FUNCTION_BLOCK HaltBehaviour IMPLEMENTS I_Task, I_Cyclic, I_Abortable, I_Object
VAR_INPUT
END_VAR
VAR_OUTPUT
END_VAR
VAR
	mcHalt : Tc2_MC2.MC_Halt;
	_Axis : REFERENCE TO Tc2_MC2.AXIS_REF;
END_VAR

{analysis -2}

METHOD Abort : HRESULT
mcHalt.Execute := FALSE;
END_METHOD

PROPERTY AxisRef : reference to Axis_Ref
GET // PUBLIC
AxisRef REF= _Axis;
END_GET
SET
_Axis REF= AxisRef;
END_SET
END_PROPERTY

PROPERTY Busy : BOOL
GET
Busy := mcHalt.Busy;
END_GET
END_PROPERTY

METHOD Cycle : HRESULT
VAR_INPUT
END_VAR
mcHalt(Axis := _Axis);
mcHalt.Execute := FALSE;
END_METHOD

PROPERTY Deceleration : MC_LREAL
GET
Deceleration := mcHalt.Deceleration;
END_GET
SET
IF Deceleration >= 0.0 THEN
	mcHalt.Deceleration := Deceleration;
END_IF
END_SET
END_PROPERTY

PROPERTY Done : BOOL
GET
Done := mcHalt.Done;
END_GET
END_PROPERTY

PROPERTY Error : BOOL
GET
Error := mcHalt.Error;
END_GET
END_PROPERTY

METHOD Execute : HRESULT
VAR_INPUT
END_VAR
IF _Axis.Status.Moving AND NOT mcHalt.Busy THEN
	Execute := S_OK;
	mcHalt.Execute := TRUE;
ELSE
	Execute := S_FALSE;
END_IF
END_METHOD

PROPERTY Jerk : MC_LREAL
GET
Jerk := mcHalt.Jerk;
END_GET
SET
IF Jerk >= 0.0 THEN
	mcHalt.Jerk := Jerk;
END_IF
END_SET
END_PROPERTY

METHOD RegisterWithParent
VAR_INPUT
	Runner	: I_HostObjects;
END_VAR
Runner.RegisterAbortable(THIS^);
Runner.RegisterCyclic(THIS^);
Runner.RegisterTask(THIS^);
END_METHOD

END_FUNCTION_BLOCK

(* stored: Version 1.1.0.1
   POU HaltBehaviour: Id {8f902aee-94bf-4385-bdcf-ca790f894752}, SpecialFunc None
   Method Abort: Id {628339b1-4bd1-432e-8277-d60f3e75db0d}
   Property AxisRef: Id {1eac54a6-2798-4751-837f-d3da316af4f3}
   Get Get: Id {b1c4cfd8-893a-485e-bd47-04ef2d23093f}
   Set Set: Id {4a81d8e2-63e1-4eb7-82a1-2f62a4d2f98c}
   Property Busy: Id {372dcfaa-8cbd-4cb0-a70e-bb4041d8e255}
   Get Get: Id {91d2b55e-e06d-4906-afcd-b4c07ffa30db}
   Method Cycle: Id {82fe1e7b-ab2b-4a89-9b59-5eb25d835959}
   Property Deceleration: Id {268ed3d1-2986-429d-85cd-2c570b60d9d7}
   Get Get: Id {907709a1-b0ba-4945-8711-6554db8f1dc0}
   Set Set: Id {502b45a2-e349-483e-b36a-b0db162a9224}
   Property Done: Id {0d4d59d1-0a33-4a35-91db-70cde82f5006}
   Get Get: Id {5c83bea7-d010-40d8-bc69-060934607785}
   Property Error: Id {3e7959eb-71d7-4ee5-89e9-4dd47b034681}
   Get Get: Id {1eaeb28a-b2d3-41f6-9d16-23d88d0071e2}
   Method Execute: Id {020a5dad-2d55-4c66-8489-dc08945209ce}
   Property Jerk: Id {bfb39f13-ace3-4f05-9305-e7d3692f5dfa}
   Get Get: Id {dfdc6efc-8e6e-48e1-a0f4-a06670061327}
   Set Set: Id {9be78a10-cc41-4de6-a2ea-3947cc380f23}
   Method RegisterWithParent: Id {761e717a-0349-45b2-b11d-2954748efbaa} *)
